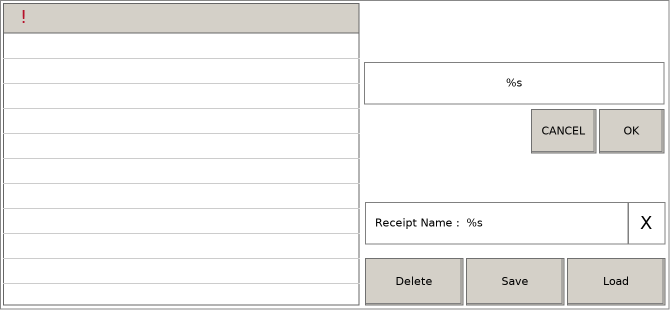
VISUALIZATION Temp_Receipt  // 670x310
VAR_IN_OUT
	stHmiRData		: ST_FB_ReceiptData;	
END_VAR
    Table (3,3 356x302), data array: stHmiRData.aReceiptFileList
        p1892666644: stHmiRData.bLoadReceipt
        p338671338: stHmiRData.bDeleteReceipt
        p2170511999: stHmiRData.nSelectedRow
        p3723444502: stHmiRData.bHmiOk
        p1218418051: stHmiRData.bHmiCancel
        p746581629: stHmiRData.sReceiptName
        p3104783080: stHmiRData.sReceiptFolder
        p2501879983: stHmiRData.bBusy
        p7306298: stHmiRData.bDone
        p1933151965: stHmiRData.bError
        p3863566920: stHmiRData.nErrorId
        p2192122294: stHmiRData.sMessage
        p400160035: stHmiRData.aReceiptFileList
        p3854506369: stHmiRData.aReceiptFileList[INDEX]
        p2232123230: RECEIPT LIST
    Rectangle (365,202 263x42), "Receipt Name : %s", text variable: stHmiRData.sReceiptName
        OnMouseClick: write the text variable via VisuDialogs.Keypad
    Button (567,258 98x47), "Load"
        tap stHmiRData.bLoadReceipt
    Button (466,258 98x47), "Save"
        tap stHmiRData.bSaveReceipt
    Button (365,258 98x47), "Delete"
        tap stHmiRData.bDeleteReceipt
    Rectangle (364,62 300x42), "%s", text variable: stHmiRData.sMessage, invisible if: stHmiRData.sMessage=''
    Button (599,109 65x44), "OK", invisible if: stHmiRData.sMessage=''
        tap stHmiRData.bHmiOk
    Button (531,109 65x44), "CANCEL", invisible if: stHmiRData.sMessage=''
        tap stHmiRData.bHmiCancel
    Rectangle (628,202 37x42), "X"
        OnMouseClick: execute { stHmiRData.sReceiptName:=''; }
    Label (7,7 33x20), "!", invisible if: stHmiRData.bError=FALSE
END_VISUALIZATION

(* stored: Version 1.1.0.1, ProductVersion 3.1.4024.12
   Visu Temp_Receipt: Id {17095dc0-1748-4203-b5fe-3539af8d7ef3} *)
